// TwinCAT 3 PLC project Untitled1
// ProgramVersion: 3.1.4023.0
// libraries:
//   Tc2_Standard, * (Beckhoff Automation GmbH)
//   Tc2_System, * (Beckhoff Automation GmbH)
//   Tc3_Module, * (Beckhoff Automation GmbH)
//   TcUnit, * (www.tcunit.org)
// project tree:
//   / PlcTask.TcTTO
//   POUs/ MAIN.TcPOU, PRG_TEST.TcPOU
//   TEST/ Example.TcPOU
// real-time tasks:
//   TASK PlcTask: cycle T#10ms, priority 20, ADS port 350

CONFIGURATION Untitled1
    RESOURCE PLC ON TwinCAT3
        TASK PlcTask(INTERVAL := T#10ms, PRIORITY := 20);
        PROGRAM MAIN WITH PlcTask : MAIN;
    END_RESOURCE
END_CONFIGURATION

// ---- POUs/MAIN.TcPOU
PROGRAM MAIN
VAR
END_VAR

PRG_TEST();

END_PROGRAM

// ---- POUs/PRG_TEST.TcPOU
PROGRAM PRG_TEST
VAR
	suite_Example : Example;
END_VAR

TcUnit.RUN();

END_PROGRAM

// ---- TEST/Example.TcPOU
FUNCTION_BLOCK Example EXTENDS tcunit.FB_TestSuite
VAR_INPUT
END_VAR
VAR_OUTPUT
END_VAR
VAR
	initWHAT				: BOOL			:= TRUE;
	initRetains 			: BOOL 			:= TRUE;
	inCopyCode 				: BOOL 			:= TRUE;
	count 					: INT 			:= 0;
	count2					: INT 			:= 0;
	currentTestNotZero		: POINTER TO FB_TestSuite;
END_VAR

IF initWHAT THEN
	initWHAT := FALSE;
	count := count + 1;
END_IF;
count2 := count2 + 1;

IF 	TcUnit.GVL_TcUnit.CurrentTestSuiteBeingCalled <> 0 THEN
	currentTestNotZero := TcUnit.GVL_TcUnit.CurrentTestSuiteBeingCalled;
END_IF

TcUnit.GVL_TcUnit.CurrentTestSuiteBeingCalled;

exampleFail();
examplePass();

// base test example for fail
METHOD exampleFail
VAR_INPUT
END_VAR
TEST('ExampleTestFail');
IF TcUnit.GVL_TcUnit.CurrentTestSuiteBeingCalled <> 0 THEN
	currentTestNotZero := TcUnit.GVL_TcUnit.CurrentTestSuiteBeingCalled;
END_IF

TcUnit.GVL_TcUnit.CurrentTestSuiteBeingCalled; 
// @TEST-RUN


// @TEST-ASSERT
AssertTrue(Condition := FALSE,
             Message := 'Test Failed Correctly');// $'emergency error code$' failed at $'diagnostic code type$'');


TEST_FINISHED();
END_METHOD

// base test example for pass
METHOD examplePass
VAR_INPUT
END_VAR
TEST('ExampleTestPass');
 
// @TEST-RUN


// @TEST-ASSERT
AssertTrue(Condition := TRUE,
             Message := 'Test should have passed');

 
TEST_FINISHED();
END_METHOD

END_FUNCTION_BLOCK
